(* Schneider Machine Expert - Basic project drum+shift bit register, file version 2.7.0.0 *)
(* ProjectInformations: Name=New project *)

HARDWARE
  Cpu 0: TM221M16R/G
  EthernetConfiguration: NetworkName=M221, IpAllocationMode=FixedAddress, IpAddress=0.0.0.0, SubnetMask=0.0.0.0
  SerialLineConfiguration: Baud=Baud19200, Parity=ParityEven, DataBits=DataBits8, StopBits=StopBits1, PhysicalMedium=PhysicalMediumRs485, TransmissionMode=TransmissionModeModbusRtu, SlaveId=1, Addressing=SlaveAddressing
  MastTask: UsePeriodScanMode=false, PeriodScan=100
  FastTask: Period=255
  CpuBehavior: StartingMode=StartAsPreviousState, AutoSaveRamOnEeprom=true, WatchdogPeriod=250

SYMBOLS  (address, symbol, comment, settings)
  %SBR0     SHIFT_BIT  [LastWritenBit=2]
  %I0.1     RESET
  %I0.2     SHIFT_LEFT
  %I0.3     SHIFT_RIGHT

POU New POU
  (* SectionNumber=1 *)

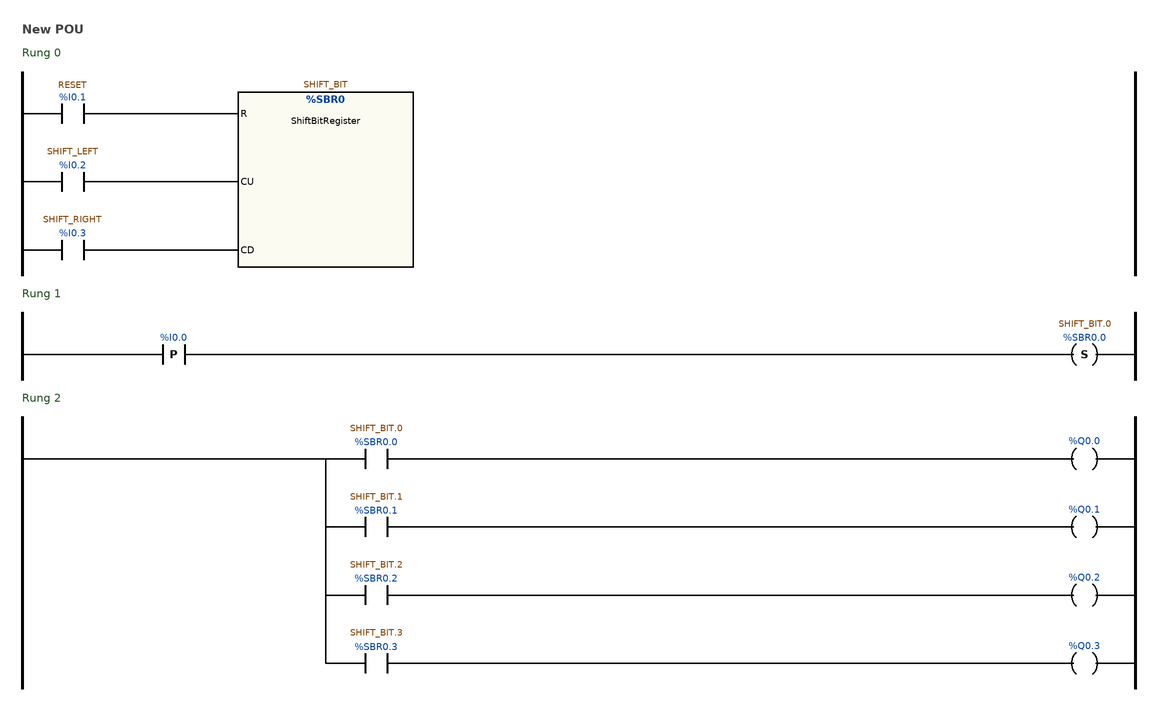

// Rung 0
  BLK %SBR0               (* SHIFT_BIT *)
  LD %I0.1                (* RESET *)
  R
  LD %I0.2                (* SHIFT_LEFT *)
  CU
  LD %I0.3                (* SHIFT_RIGHT *)
  CD
  END_BLK
  // as ST:
  //   SHIFT_BIT(R := RESET, CU := SHIFT_LEFT, CD := SHIFT_RIGHT);

// Rung 1
  LDR %I0.0
  S %SBR0.0
  // as ST:
  //   IF RISING(%I0.0) THEN %SBR0.0 := TRUE; END_IF;

// Rung 2
  LD 1
  MPS
  AND %SBR0.0
  ST %Q0.0
  MRD
  AND %SBR0.1
  ST %Q0.1
  MRD
  AND %SBR0.2
  ST %Q0.2
  MPP
  AND %SBR0.3
  ST %Q0.3
  // as ST:
  //   %Q0.0 := %SBR0.0;
  //   %Q0.1 := %SBR0.1;
  //   %Q0.2 := %SBR0.2;
  //   %Q0.3 := %SBR0.3;
